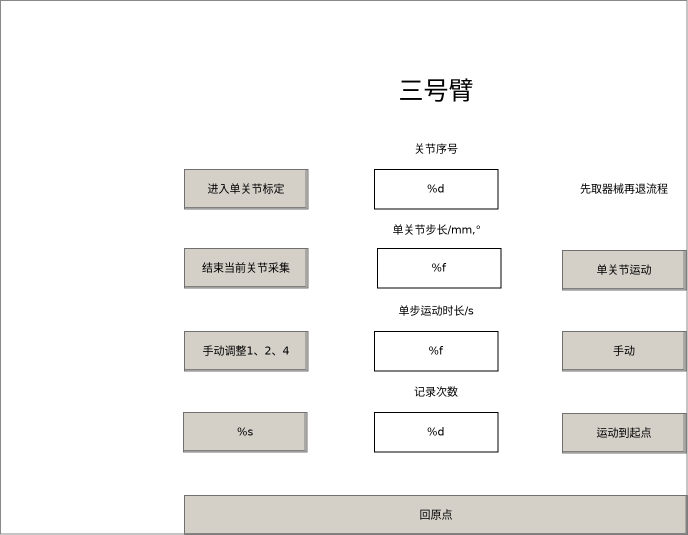
VISUALIZATION kineCali_a3  // 688x535
    Button (184,169 124x40), "进入单关节标定", colour toggle: g_singleJntTest.m_enterSingleJntTestMode[3]
        toggle g_singleJntTest.m_enterSingleJntTestMode[3]
    Button (562,331 124x40), "手动", colour toggle: g_singleJntTest.m_manualAdjustFlag
    Button (562,413 124x40), "运动到起点", colour toggle: g_singleJntTest.m_move2StartFlag
    Rectangle (374,412 124x40), "%d", text variable: g_singleJntTest.m_dataRecordCount[3]
        OnMouseClick: write the text variable via Default, min 0, max 1000
    Label (362,210 150x40), "单关节步长/mm,°"
    Button (562,250 124x40), "单关节运动", colour toggle: g_singleJntTest.m_singleJntFlag
    Label (361,129 150x40), "关节序号"
    Rectangle (377,248 124x40), "%f", text variable: g_singleJntTest.m_jntStep
        OnMouseClick: write the text variable via Default, min 0
    Button (183,412 124x40), "%s", text variable: g_singleJntTest.m_dataRecordText, colour toggle: g_singleJntTest.m_dataRecordFlag[3]
        tap g_singleJntTest.m_dataRecordFlag[3]
    Rectangle (374,169 124x40), "%d", text variable: g_singleJntTest.m_kineCaliJntIdx
        OnMouseClick: write the text variable via Default, min 1, max 8
    Button (184,495 504x40), "回原点", colour toggle: g_singleJntTest.m_return2OriginFlag
    Rectangle (374,331 124x40), "%f", text variable: g_singleJntTest.m_EndT
        OnMouseClick: write the text variable via Default, min 0, max 100
    Label (361,291 150x40), "单步运动时长/s"
    Label (361,372 150x40), "记录次数"
    Label (361,69 150x43), "三号臂"
    Button (184,248 124x40), "结束当前关节采集", colour toggle: g_singleJntTest.m_manualEndFlag
        toggle g_singleJntTest.m_manualEndFlag
    Button (184,331 124x40), "手动调整1、2、4", colour toggle: g_singleJntTest.m_manual124StartFlag
        toggle g_singleJntTest.m_manual124StartFlag
    Label (562,169 124x40), "先取器械再退流程"
END_VISUALIZATION

(* stored: Version 1.1.0.1, ProductVersion 3.1.4024.11
   Visu kineCali_a3: Id {40fe9613-1321-43d0-a69c-38fca4b72e7f} *)
